(* IEC 61131-3 sources: StandardFunctions/iec61131-st (part 2) *)

(* ---- time_extra_functions.st ---- *)
(********************
*
* Concatenates DATE and TOD to DT
*
*********************)
@EXTERNAL
FUNCTION CONCAT_DATE_TOD : DT
VAR_INPUT
	date_input : DATE;
	tod_input : TOD;
END_VAR
END_FUNCTION

(********************
*
* Concatenates DATE and LTOD to DT
*
*********************)
FUNCTION CONCAT_DATE_LTOD : DT
VAR_INPUT
	date_input : DATE;
	tod_input : LTOD;
END_VAR
	CONCAT_DATE_LTOD := CONCAT_DATE_TOD(date_input, tod_input);
END_FUNCTION

(********************
*
* Concatenates year, month and day of type ANY_INT to DATE
*
*********************)
@EXTERNAL
FUNCTION CONCAT_DATE <T: ANY_INT> : DATE
VAR_INPUT
	year : T;
	month : T;
	day : T;
END_VAR
END_FUNCTION

(********************
*
* Concatenates hour, minute, second, millisecond of type ANY_INT to TOD
*
*********************)
@EXTERNAL
FUNCTION CONCAT_TOD <T: ANY_INT> : TOD
VAR_INPUT
	hour : T;
	minute : T;
	second : T;
	millisecond : T;
END_VAR
END_FUNCTION

(********************
*
* Concatenates hour, minute, second, millisecond of type ANY_INT to LTOD
*
*********************)
FUNCTION CONCAT_LTOD <T: ANY_INT> : LTOD
VAR_INPUT
	hour : T;
	minute : T;
	second : T;
	millisecond : T;
END_VAR
END_FUNCTION

(* Specialized implementation of CONCAT_LTOD for SINT *)
FUNCTION CONCAT_LTOD__SINT : LTOD
VAR_INPUT
	hour : SINT;
	minute : SINT;
	second : SINT;
	millisecond : SINT;
END_VAR
	CONCAT_LTOD__SINT := CONCAT_TOD(hour, minute, second, millisecond);
END_FUNCTION

(* Specialized implementation of CONCAT_LTOD for USINT *)
FUNCTION CONCAT_LTOD__USINT : LTOD
VAR_INPUT
	hour : USINT;
	minute : USINT;
	second : USINT;
	millisecond : USINT;
END_VAR
	CONCAT_LTOD__USINT := CONCAT_TOD(hour, minute, second, millisecond);
END_FUNCTION

(* Specialized implementation of CONCAT_LTOD for INT *)
FUNCTION CONCAT_LTOD__INT : LTOD
VAR_INPUT
	hour : INT;
	minute : INT;
	second : INT;
	millisecond : INT;
END_VAR
	CONCAT_LTOD__INT := CONCAT_TOD(hour, minute, second, millisecond);
END_FUNCTION

(* Specialized implementation of CONCAT_LTOD for UINT *)
FUNCTION CONCAT_LTOD__UINT : LTOD
VAR_INPUT
	hour : UINT;
	minute : UINT;
	second : UINT;
	millisecond : UINT;
END_VAR
	CONCAT_LTOD__UINT := CONCAT_TOD(hour, minute, second, millisecond);
END_FUNCTION

(* Specialized implementation of CONCAT_LTOD for DINT *)
FUNCTION CONCAT_LTOD__DINT : LTOD
VAR_INPUT
	hour : DINT;
	minute : DINT;
	second : DINT;
	millisecond : DINT;
END_VAR
	CONCAT_LTOD__DINT := CONCAT_TOD(hour, minute, second, millisecond);
END_FUNCTION

(* Specialized implementation of CONCAT_LTOD for UDINT *)
FUNCTION CONCAT_LTOD__UDINT : LTOD
VAR_INPUT
	hour : UDINT;
	minute : UDINT;
	second : UDINT;
	millisecond : UDINT;
END_VAR
	CONCAT_LTOD__UDINT := CONCAT_TOD(hour, minute, second, millisecond);
END_FUNCTION

(* Specialized implementation of CONCAT_LTOD for LINT *)
FUNCTION CONCAT_LTOD__LINT : LTOD
VAR_INPUT
	hour : LINT;
	minute : LINT;
	second : LINT;
	millisecond : LINT;
END_VAR
	CONCAT_LTOD__LINT := CONCAT_TOD(hour, minute, second, millisecond);
END_FUNCTION

(* Specialized implementation of CONCAT_LTOD for ULINT *)
FUNCTION CONCAT_LTOD__ULINT : LTOD
VAR_INPUT
	hour : ULINT;
	minute : ULINT;
	second : ULINT;
	millisecond : ULINT;
END_VAR
	CONCAT_LTOD__ULINT := CONCAT_TOD(hour, minute, second, millisecond);
END_FUNCTION

(********************
*
* Concatenates year, month, day, hour, minute, second, millisecond of type ANY_INT to DT
*
*********************)
FUNCTION CONCAT_DT <T: ANY_INT> : DT
VAR_INPUT
	year : T;
	month : T;
	day : T;
	hour : T;
	minute : T;
	second : T;
	millisecond : T;
END_VAR
END_FUNCTION

(* Specialized implementation of CONCAT_DT for INT *)
FUNCTION CONCAT_DT__INT : DT
VAR_INPUT
	year : INT;
	month : INT;
	day : INT;
	hour : INT;
	minute : INT;
	second : INT;
	millisecond : INT;
END_VAR
	CONCAT_DT__INT := CONCAT_DATE_TOD(CONCAT_DATE(year, month, day), CONCAT_TOD(hour, minute, second, millisecond));
END_FUNCTION

(* Specialized implementation of CONCAT_DT for UINT *)
FUNCTION CONCAT_DT__UINT : DT
VAR_INPUT
	year : UINT;
	month : UINT;
	day : UINT;
	hour : UINT;
	minute : UINT;
	second : UINT;
	millisecond : UINT;
END_VAR
	CONCAT_DT__UINT := CONCAT_DATE_TOD(CONCAT_DATE(year, month, day), CONCAT_TOD(hour, minute, second, millisecond));
END_FUNCTION

(* Specialized implementation of CONCAT_DT for DINT *)
FUNCTION CONCAT_DT__DINT : DT
VAR_INPUT
	year : DINT;
	month : DINT;
	day : DINT;
	hour : DINT;
	minute : DINT;
	second : DINT;
	millisecond : DINT;
END_VAR
	CONCAT_DT__DINT := CONCAT_DATE_TOD(CONCAT_DATE(year, month, day), CONCAT_TOD(hour, minute, second, millisecond));
END_FUNCTION

(* Specialized implementation of CONCAT_DT for UDINT *)
FUNCTION CONCAT_DT__UDINT : DT
VAR_INPUT
	year : UDINT;
	month : UDINT;
	day : UDINT;
	hour : UDINT;
	minute : UDINT;
	second : UDINT;
	millisecond : UDINT;
END_VAR
	CONCAT_DT__UDINT := CONCAT_DATE_TOD(CONCAT_DATE(year, month, day), CONCAT_TOD(hour, minute, second, millisecond));
END_FUNCTION

(* Specialized implementation of CONCAT_DT for LINT *)
FUNCTION CONCAT_DT__LINT : DT
VAR_INPUT
	year : LINT;
	month : LINT;
	day : LINT;
	hour : LINT;
	minute : LINT;
	second : LINT;
	millisecond : LINT;
END_VAR
	CONCAT_DT__LINT := CONCAT_DATE_TOD(CONCAT_DATE(year, month, day), CONCAT_TOD(hour, minute, second, millisecond));
END_FUNCTION

(* Specialized implementation of CONCAT_DT for ULINT *)
FUNCTION CONCAT_DT__ULINT : DT
VAR_INPUT
	year : ULINT;
	month : ULINT;
	day : ULINT;
	hour : ULINT;
	minute : ULINT;
	second : ULINT;
	millisecond : ULINT;
END_VAR
	CONCAT_DT__ULINT := CONCAT_DATE_TOD(CONCAT_DATE(year, month, day), CONCAT_TOD(hour, minute, second, millisecond));
END_FUNCTION

(********************
*
* Concatenates year, month, day, hour, minute, second, millisecond of type ANY_INT to LDT
*
*********************)
FUNCTION CONCAT_LDT <T: ANY_INT> : LDT
VAR_INPUT
	year : T;
	month : T;
	day : T;
	hour : T;
	minute : T;
	second : T;
	millisecond : T;
END_VAR
END_FUNCTION

(* Specialized implementation of CONCAT_LDT for INT *)
FUNCTION CONCAT_LDT__INT : LDT
VAR_INPUT
	year : INT;
	month : INT;
	day : INT;
	hour : INT;
	minute : INT;
	second : INT;
	millisecond : INT;
END_VAR
	CONCAT_LDT__INT := CONCAT_DATE_LTOD(CONCAT_DATE(year, month, day), CONCAT_LTOD(hour, minute, second, millisecond));
END_FUNCTION

(* Specialized implementation of CONCAT_LDT for UINT *)
FUNCTION CONCAT_LDT__UINT : LDT
VAR_INPUT
	year : UINT;
	month : UINT;
	day : UINT;
	hour : UINT;
	minute : UINT;
	second : UINT;
	millisecond : UINT;
END_VAR
	CONCAT_LDT__UINT := CONCAT_DATE_LTOD(CONCAT_DATE(year, month, day), CONCAT_LTOD(hour, minute, second, millisecond));
END_FUNCTION

(* Specialized implementation of CONCAT_LDT for DINT *)
FUNCTION CONCAT_LDT__DINT : LDT
VAR_INPUT
	year : DINT;
	month : DINT;
	day : DINT;
	hour : DINT;
	minute : DINT;
	second : DINT;
	millisecond : DINT;
END_VAR
	CONCAT_LDT__DINT := CONCAT_DATE_LTOD(CONCAT_DATE(year, month, day), CONCAT_LTOD(hour, minute, second, millisecond));
END_FUNCTION

(* Specialized implementation of CONCAT_LDT for UDINT *)
FUNCTION CONCAT_LDT__UDINT : LDT
VAR_INPUT
	year : UDINT;
	month : UDINT;
	day : UDINT;
	hour : UDINT;
	minute : UDINT;
	second : UDINT;
	millisecond : UDINT;
END_VAR
	CONCAT_LDT__UDINT := CONCAT_DATE_LTOD(CONCAT_DATE(year, month, day), CONCAT_LTOD(hour, minute, second, millisecond));
END_FUNCTION

(* Specialized implementation of CONCAT_LDT for LINT *)
FUNCTION CONCAT_LDT__LINT : LDT
VAR_INPUT
	year : LINT;
	month : LINT;
	day : LINT;
	hour : LINT;
	minute : LINT;
	second : LINT;
	millisecond : LINT;
END_VAR
	CONCAT_LDT__LINT := CONCAT_DATE_LTOD(CONCAT_DATE(year, month, day), CONCAT_LTOD(hour, minute, second, millisecond));
END_FUNCTION

(* Specialized implementation of CONCAT_LDT for ULINT *)
FUNCTION CONCAT_LDT__ULINT : LDT
VAR_INPUT
	year : ULINT;
	month : ULINT;
	day : ULINT;
	hour : ULINT;
	minute : ULINT;
	second : ULINT;
	millisecond : ULINT;
END_VAR
	CONCAT_LDT__ULINT := CONCAT_DATE_LTOD(CONCAT_DATE(year, month, day), CONCAT_LTOD(hour, minute, second, millisecond));
END_FUNCTION

(********************
*
* Splits DATE into year, month, day of type ANY_INT
*
*********************)
FUNCTION SPLIT_DATE <T: ANY_INT> : INT
VAR_INPUT
	in : DATE;
END_VAR
VAR_OUTPUT
	year : T;
	month : T;
	day : T;
END_VAR
END_FUNCTION

(* Specialized implementation of SPLIT_DATE for INT *)
@EXTERNAL
FUNCTION SPLIT_DATE__INT : INT
VAR_INPUT
	in : DATE;
END_VAR
VAR_OUTPUT
	year : INT;
	month : INT;
	day : INT;
END_VAR
END_FUNCTION

(* Specialized implementation of SPLIT_DATE for UINT *)
@EXTERNAL
FUNCTION SPLIT_DATE__UINT : INT
VAR_INPUT
	in : DATE;
END_VAR
VAR_OUTPUT
	year : UINT;
	month : UINT;
	day : UINT;
END_VAR
END_FUNCTION

(* Specialized implementation of SPLIT_DATE for DINT *)
@EXTERNAL
FUNCTION SPLIT_DATE__DINT : INT
VAR_INPUT
	in : DATE;
END_VAR
VAR_OUTPUT
	year : DINT;
	month : DINT;
	day : DINT;
END_VAR
END_FUNCTION

(* Specialized implementation of SPLIT_DATE for UDINT *)
@EXTERNAL
FUNCTION SPLIT_DATE__UDINT : INT
VAR_INPUT
	in : DATE;
END_VAR
VAR_OUTPUT
	year : UDINT;
	month : UDINT;
	day : UDINT;
END_VAR
END_FUNCTION

(* Specialized implementation of SPLIT_DATE for LINT *)
@EXTERNAL
FUNCTION SPLIT_DATE__LINT : INT
VAR_INPUT
	in : DATE;
END_VAR
VAR_OUTPUT
	year : LINT;
	month : LINT;
	day : LINT;
END_VAR
END_FUNCTION

(* Specialized implementation of SPLIT_DATE for ULINT *)
@EXTERNAL
FUNCTION SPLIT_DATE__ULINT : INT
VAR_INPUT
	in : DATE;
END_VAR
VAR_OUTPUT
	year : ULINT;
	month : ULINT;
	day : ULINT;
END_VAR
END_FUNCTION

(********************
*
* Splits TOD into hour, minute, second, millisecond of type ANY_INT
*
*********************)
FUNCTION SPLIT_TOD <T: ANY_INT> : INT
VAR_INPUT
	in : TOD;
END_VAR
VAR_OUTPUT
	hour : T;
	minute : T;
	second : T;
	millisecond : T;
END_VAR
END_FUNCTION

(* Specialized implementation of SPLIT_TOD for INT *)
@EXTERNAL
FUNCTION SPLIT_TOD__INT : INT
VAR_INPUT
	in : TOD;
END_VAR
VAR_OUTPUT
	hour : INT;
	minute : INT;
	second : INT;
	millisecond : INT;
END_VAR
END_FUNCTION

(* Specialized implementation of SPLIT_TOD for UINT *)
@EXTERNAL
FUNCTION SPLIT_TOD__UINT : INT
VAR_INPUT
	in : TOD;
END_VAR
VAR_OUTPUT
	hour : UINT;
	minute : UINT;
	second : UINT;
	millisecond : UINT;
END_VAR
END_FUNCTION

(* Specialized implementation of SPLIT_TOD for DINT *)
@EXTERNAL
FUNCTION SPLIT_TOD__DINT : INT
VAR_INPUT
	in : TOD;
END_VAR
VAR_OUTPUT
	hour : DINT;
	minute : DINT;
	second : DINT;
	millisecond : DINT;
END_VAR
END_FUNCTION

(* Specialized implementation of SPLIT_TOD for UDINT *)
@EXTERNAL
FUNCTION SPLIT_TOD__UDINT : INT
VAR_INPUT
	in : TOD;
END_VAR
VAR_OUTPUT
	hour : UDINT;
	minute : UDINT;
	second : UDINT;
	millisecond : UDINT;
END_VAR
END_FUNCTION

(* Specialized implementation of SPLIT_TOD for LINT *)
@EXTERNAL
FUNCTION SPLIT_TOD__LINT : INT
VAR_INPUT
	in : TOD;
END_VAR
VAR_OUTPUT
	hour : LINT;
	minute : LINT;
	second : LINT;
	millisecond : LINT;
END_VAR
END_FUNCTION

(* Specialized implementation of SPLIT_TOD for ULINT *)
@EXTERNAL
FUNCTION SPLIT_TOD__ULINT : INT
VAR_INPUT
	in : TOD;
END_VAR
VAR_OUTPUT
	hour : ULINT;
	minute : ULINT;
	second : ULINT;
	millisecond : ULINT;
END_VAR
END_FUNCTION

(********************
*
* Splits LTOD into hour, minute, second, millisecond of type ANY_INT
*
*********************)
FUNCTION SPLIT_LTOD <T: ANY_INT> : INT
VAR_INPUT
	in : LTOD;
END_VAR
VAR_OUTPUT
	hour : T;
	minute : T;
	second : T;
	millisecond : T;
END_VAR
END_FUNCTION

(* Specialized implementation of SPLIT_LTOD for INT *)
FUNCTION SPLIT_LTOD__INT : INT
VAR_INPUT
	in : LTOD;
END_VAR
VAR_OUTPUT
	hour : INT;
	minute : INT;
	second : INT;
	millisecond : INT;
END_VAR
	SPLIT_LTOD__INT := SPLIT_TOD__INT(in, hour, minute, second, millisecond);
END_FUNCTION

(* Specialized implementation of SPLIT_LTOD for UINT *)
FUNCTION SPLIT_LTOD__UINT : INT
VAR_INPUT
	in : LTOD;
END_VAR
VAR_OUTPUT
	hour : UINT;
	minute : UINT;
	second : UINT;
	millisecond : UINT;
END_VAR
	SPLIT_LTOD__UINT := SPLIT_TOD__UINT(in, hour, minute, second, millisecond);
END_FUNCTION

(* Specialized implementation of SPLIT_LTOD for DINT *)
FUNCTION SPLIT_LTOD__DINT : INT
VAR_INPUT
	in : LTOD;
END_VAR
VAR_OUTPUT
	hour : DINT;
	minute : DINT;
	second : DINT;
	millisecond : DINT;
END_VAR
	SPLIT_LTOD__DINT := SPLIT_TOD__DINT(in, hour, minute, second, millisecond);
END_FUNCTION

(* Specialized implementation of SPLIT_LTOD for UDINT *)
FUNCTION SPLIT_LTOD__UDINT : INT
VAR_INPUT
	in : LTOD;
END_VAR
VAR_OUTPUT
	hour : UDINT;
	minute : UDINT;
	second : UDINT;
	millisecond : UDINT;
END_VAR
	SPLIT_LTOD__UDINT := SPLIT_TOD__UDINT(in, hour, minute, second, millisecond);
END_FUNCTION

(* Specialized implementation of SPLIT_LTOD for LINT *)
FUNCTION SPLIT_LTOD__LINT : INT
VAR_INPUT
	in : LTOD;
END_VAR
VAR_OUTPUT
	hour : LINT;
	minute : LINT;
	second : LINT;
	millisecond : LINT;
END_VAR
	SPLIT_LTOD__LINT := SPLIT_TOD__LINT(in, hour, minute, second, millisecond);
END_FUNCTION

(* Specialized implementation of SPLIT_LTOD for ULINT *)
FUNCTION SPLIT_LTOD__ULINT : INT
VAR_INPUT
	in : LTOD;
END_VAR
VAR_OUTPUT
	hour : ULINT;
	minute : ULINT;
	second : ULINT;
	millisecond : ULINT;
END_VAR
	SPLIT_LTOD__ULINT := SPLIT_TOD__ULINT(in, hour, minute, second, millisecond);
END_FUNCTION

(********************
*
* Splits DT into year, month, day, hour, minute, second, millisecond of type ANY_INT
*
*********************)
FUNCTION SPLIT_DT <T: ANY_INT> : INT
VAR_INPUT
	in : DT;
END_VAR
VAR_OUTPUT
	year : T;
	month : T;
	day : T;
	hour : T;
	minute : T;
	second : T;
	millisecond : T;
END_VAR
END_FUNCTION

(* Specialized implementation of SPLIT_DT for INT *)
@EXTERNAL
FUNCTION SPLIT_DT__INT : INT
VAR_INPUT
	in : DT;
END_VAR
VAR_OUTPUT
	year : INT;
	month : INT;
	day : INT;
	hour : INT;
	minute : INT;
	second : INT;
	millisecond : INT;
END_VAR
END_FUNCTION

(* Specialized implementation of SPLIT_DT for UINT *)
@EXTERNAL
FUNCTION SPLIT_DT__UINT : INT
VAR_INPUT
	in : DT;
END_VAR
VAR_OUTPUT
	year : UINT;
	month : UINT;
	day : UINT;
	hour : UINT;
	minute : UINT;
	second : UINT;
	millisecond : UINT;
END_VAR
END_FUNCTION

(* Specialized implementation of SPLIT_DT for DINT *)
@EXTERNAL
FUNCTION SPLIT_DT__DINT : INT
VAR_INPUT
	in : DT;
END_VAR
VAR_OUTPUT
	year : DINT;
	month : DINT;
	day : DINT;
	hour : DINT;
	minute : DINT;
	second : DINT;
	millisecond : DINT;
END_VAR
END_FUNCTION

(* Specialized implementation of SPLIT_DT for UDINT *)
@EXTERNAL
FUNCTION SPLIT_DT__UDINT : INT
VAR_INPUT
	in : DT;
END_VAR
VAR_OUTPUT
	year : UDINT;
	month : UDINT;
	day : UDINT;
	hour : UDINT;
	minute : UDINT;
	second : UDINT;
	millisecond : UDINT;
END_VAR
END_FUNCTION

(* Specialized implementation of SPLIT_DT for LINT *)
@EXTERNAL
FUNCTION SPLIT_DT__LINT : INT
VAR_INPUT
	in : DT;
END_VAR
VAR_OUTPUT
	year : LINT;
	month : LINT;
	day : LINT;
	hour : LINT;
	minute : LINT;
	second : LINT;
	millisecond : LINT;
END_VAR
END_FUNCTION

(* Specialized implementation of SPLIT_DT for ULINT *)
@EXTERNAL
FUNCTION SPLIT_DT__ULINT : INT
VAR_INPUT
	in : DT;
END_VAR
VAR_OUTPUT
	year : ULINT;
	month : ULINT;
	day : ULINT;
	hour : ULINT;
	minute : ULINT;
	second : ULINT;
	millisecond : ULINT;
END_VAR
END_FUNCTION

(********************
*
* Splits LDT into year, month, day, hour, minute, second, millisecond of type ANY_INT
*
*********************)
FUNCTION SPLIT_LDT <T: ANY_INT> : INT
VAR_INPUT
	in : LDT;
END_VAR
VAR_OUTPUT
	year : T;
	month : T;
	day : T;
	hour : T;
	minute : T;
	second : T;
	millisecond : T;
END_VAR
END_FUNCTION

(* Specialized implementation of SPLIT_LDT for INT *)
@EXTERNAL
FUNCTION SPLIT_LDT__INT : INT
VAR_INPUT
	in : LDT;
END_VAR
VAR_OUTPUT
	year : INT;
	month : INT;
	day : INT;
	hour : INT;
	minute : INT;
	second : INT;
	millisecond : INT;
END_VAR
	SPLIT_LDT__INT := SPLIT_DT__INT(in, year, month, day, hour, minute, second, millisecond);
END_FUNCTION

(* Specialized implementation of SPLIT_LDT for UINT *)
@EXTERNAL
FUNCTION SPLIT_LDT__UINT : INT
VAR_INPUT
	in : LDT;
END_VAR
VAR_OUTPUT
	year : UINT;
	month : UINT;
	day : UINT;
	hour : UINT;
	minute : UINT;
	second : UINT;
	millisecond : UINT;
END_VAR
	SPLIT_LDT__UINT := SPLIT_DT__UINT(in, year, month, day, hour, minute, second, millisecond);
END_FUNCTION

(* Specialized implementation of SPLIT_LDT for DINT *)
@EXTERNAL
FUNCTION SPLIT_LDT__DINT : INT
VAR_INPUT
	in : LDT;
END_VAR
VAR_OUTPUT
	year : DINT;
	month : DINT;
	day : DINT;
	hour : DINT;
	minute : DINT;
	second : DINT;
	millisecond : DINT;
END_VAR
	SPLIT_LDT__DINT := SPLIT_DT__DINT(in, year, month, day, hour, minute, second, millisecond);
END_FUNCTION

(* Specialized implementation of SPLIT_LDT for UDINT *)
@EXTERNAL
FUNCTION SPLIT_LDT__UDINT : INT
VAR_INPUT
	in : LDT;
END_VAR
VAR_OUTPUT
	year : UDINT;
	month : UDINT;
	day : UDINT;
	hour : UDINT;
	minute : UDINT;
	second : UDINT;
	millisecond : UDINT;
END_VAR
	SPLIT_LDT__UDINT := SPLIT_DT__UDINT(in, year, month, day, hour, minute, second, millisecond);
END_FUNCTION

(* Specialized implementation of SPLIT_LDT for LINT *)
@EXTERNAL
FUNCTION SPLIT_LDT__LINT : INT
VAR_INPUT
	in : LDT;
END_VAR
VAR_OUTPUT
	year : LINT;
	month : LINT;
	day : LINT;
	hour : LINT;
	minute : LINT;
	second : LINT;
	millisecond : LINT;
END_VAR
	SPLIT_LDT__LINT := SPLIT_DT__LINT(in, year, month, day, hour, minute, second, millisecond);
END_FUNCTION

(* Specialized implementation of SPLIT_LDT for ULINT *)
@EXTERNAL
FUNCTION SPLIT_LDT__ULINT : INT
VAR_INPUT
	in : LDT;
END_VAR
VAR_OUTPUT
	year : ULINT;
	month : ULINT;
	day : ULINT;
	hour : ULINT;
	minute : ULINT;
	second : ULINT;
	millisecond : ULINT;
END_VAR
	SPLIT_LDT__ULINT := SPLIT_DT__ULINT(in, year, month, day, hour, minute, second, millisecond);
END_FUNCTION

(********************
*
* Returns day of week form given DATE in SINT
* 0 -> sunday, 1 -> monday, ..., 6 -> saturday
*
*********************)
@EXTERNAL
FUNCTION DAY_OF_WEEK : SINT
VAR_INPUT
	in : DATE;
END_VAR
END_FUNCTION

(* ---- validation.st ---- *)
(******************************************************************************
Description: Validation function for ANY_REAL
Input:
  - IN: ANY_REAL
Return:
  - FALSE: If input is Not-a-Number(NaN) or infinite(+Inf, -Inf)
  - TRUE: Otherwise
******************************************************************************)
FUNCTION IS_VALID <T: ANY_REAL> : BOOL
VAR_INPUT
	IN : T;
END_VAR
END_FUNCTION

(******************************************************************************
Description: Validation function for ANY_BIT
Validate if the binary representation of the input
would result in a valid BCD representation
Input:
  - IN: ANY_BIT
Return:
  - TRUE: The value of each 4bits representet digit must be between 0-9
  - FALSE: If the value of any 4bits representet digit is higher than 9
******************************************************************************)
FUNCTION IS_VALID_BCD <T: ANY_BIT> : BOOL
VAR_INPUT
	IN : T;
END_VAR
END_FUNCTION

(* ---- bistable_functionblocks.st ---- *)
(******************************************************************************
Description: Bistable function, set dominant
Input:
  - SET1: Dominant input of bistable function.
  - RESET: input of bistable function.
Output:
  - Q1: Result of Bistable function.
Return: Output is used as return
******************************************************************************)
{external}
FUNCTION_BLOCK SR
VAR_INPUT
	SET1: BOOL;
	RESET: BOOL;
END_VAR
VAR_OUTPUT
	Q1: BOOL;
END_VAR
END_FUNCTION_BLOCK

(******************************************************************************
Description: Bistable function, reset dominant.
Input:
  - SET: Bistable input
  - RESET1: Dominmant bistable input.
Output:
  - Q1: Result of bistable function
Return: Output variable used as return value.
******************************************************************************)
{external}
FUNCTION_BLOCK RS
VAR_INPUT
	SET: 	BOOL;
	RESET1: BOOL;
END_VAR
VAR_OUTPUT
	Q1:		BOOL;
END_VAR
END_FUNCTION_BLOCK

(* ---- counters.st ---- *)
(******************************************************************************
Description: Counter up
Input:
  - CU: Count up
  - R: Reset counter to 0
  - PV: Counter limit
Output:
  - Q: Counter reached limit
  - CV: Current counter value
Return: Output is used as return value
******************************************************************************)
{external}
FUNCTION_BLOCK CTU_INT
VAR_INPUT
	CU : BOOL;
	R : BOOL;
	PV : INT;
END_VAR
VAR_OUTPUT
	Q : BOOL;
	CV : INT;
END_VAR
VAR
	M : BOOL;
END_VAR
END_FUNCTION_BLOCK

(******************************************************************************
Description: Counter up
Input:
  - CU: Count up
  - R: Reset counter to 0
  - PV: Counter limit
Output:
  - Q: Counter reached limit
  - CV: Current counter value
Return: Output is used as return value
******************************************************************************)
{external}
FUNCTION_BLOCK CTU_DINT
VAR_INPUT
	CU : BOOL;
	R : BOOL;
	PV : DINT;
END_VAR
VAR_OUTPUT
	Q : BOOL;
	CV : DINT;
END_VAR
VAR
	M : BOOL;
END_VAR
END_FUNCTION_BLOCK

(******************************************************************************
Description: Counter up
Input:
  - CU: Count up
  - R: Reset counter to 0
  - PV: Counter limit
Output:
  - Q: Counter reached limit
  - CV: Current counter value
Return: Output is used as return value
******************************************************************************)
{external}
FUNCTION_BLOCK CTU_UDINT
VAR_INPUT
	CU : BOOL;
	R : BOOL;
	PV : UDINT;
END_VAR
VAR_OUTPUT
	Q : BOOL;
	CV : UDINT;
END_VAR
VAR
	M : BOOL;
END_VAR
END_FUNCTION_BLOCK

(******************************************************************************
Description: Counter up
Input:
  - CU: Count up
  - R: Reset counter to 0
  - PV: Counter limit
Output:
  - Q: Counter reached limit
  - CV: Current counter value
Return: Output is used as return value
******************************************************************************)
{external}
FUNCTION_BLOCK CTU_LINT
VAR_INPUT
	CU : BOOL;
	R : BOOL;
	PV : LINT;
END_VAR
VAR_OUTPUT
	Q : BOOL;
	CV : LINT;
END_VAR
VAR
	M : BOOL;
END_VAR
END_FUNCTION_BLOCK

(******************************************************************************
Description: Counter up
Input:
  - CU: Count up
  - R: Reset counter to 0
  - PV: Counter limit
Output:
  - Q: Counter reached limit
  - CV: Current counter value
Return: Output is used as return value
******************************************************************************)
{external}
FUNCTION_BLOCK CTU_ULINT
VAR_INPUT
	CU : BOOL;
	R : BOOL;
	PV : ULINT;
END_VAR
VAR_OUTPUT
	Q : BOOL;
	CV : ULINT;
END_VAR
VAR
	M : BOOL;
END_VAR
END_FUNCTION_BLOCK

(* ---- timers.st ---- *)
{external}
(******************************************************************************
Description: Timer Pulse
Input:
  - IN: Trigger for Start of the Signal
  - PT: The length of the High-Signal
Output:
  - Q: The pulse
  - ET: The current phase of the High-Signal
Return: Output variables are used for return.
******************************************************************************)
FUNCTION_BLOCK TP
    VAR_INPUT
        IN : BOOL;
        PT : TIME;
    END_VAR
    VAR_OUTPUT
        Q  : BOOL;
        ET : TIME;
    END_VAR
    VAR
        __signal__ : BOOL; (* Value representing the internal signal *)
        __BUFFER__ : ARRAY[1..24] OF BYTE; (* Buffer used for internal implementation *)
    END_VAR
END_FUNCTION_BLOCK

{external}
(******************************************************************************
Description: Timer Pulse
Input:
  - IN: Trigger for Start of the Signal
  - PT: The length of the High-Signal
Output:
  - Q: The pulse
  - ET: The current phase of the High-Signal
Return: Output variables are used for return.
******************************************************************************)
FUNCTION_BLOCK TP_TIME
    VAR_INPUT
        IN : BOOL;
        PT : TIME;
    END_VAR
    VAR_OUTPUT
        Q  : BOOL;
        ET : TIME;
    END_VAR
    VAR
      __signal__ : BOOL; (* Value representing the internal signal *)
      __BUFFER__ : ARRAY[1..24] OF BYTE; (* Buffer used for internal implementation *)
    END_VAR
END_FUNCTION_BLOCK

{external}
(******************************************************************************
Description: Timer Pulse
Input:
  - IN: Trigger for Start of the Signal
  - PT: The length of the High-Signal
Output:
  - Q: The pulse
  - ET: The current phase of the High-Signal
Return: Output variables are used for return.
******************************************************************************)
FUNCTION_BLOCK TP_LTIME
    VAR_INPUT
        IN : BOOL;
        PT : TIME;
    END_VAR
    VAR_OUTPUT
        Q  : BOOL;
        ET : LTIME;
    END_VAR
    VAR
        __signal__ : BOOL; (* Value representing the internal signal *)
        __BUFFER__ : ARRAY[1..24] OF BYTE; (* Buffer used for internal implementation *)
    END_VAR
END_FUNCTION_BLOCK

{external}
(******************************************************************************
Description: Timer on delay.
Input:
  - IN: Starts timer with rising edge, resets timer with falling edge
  - PT: Time to pass, before Q is set
Output:
  - Q: Is TRUE, PT seconds after IN had a rising edge
  - ET: Elapsed time
Return: Output variables are used for return.
******************************************************************************)
FUNCTION_BLOCK TON
VAR_INPUT
	IN: BOOL;
	PT: TIME;
END_VAR
VAR_OUTPUT
	Q: BOOL;
	ET: TIME;
END_VAR
VAR
  __signal__ : BOOL; (* Value representing the internal signal *)
  __BUFFER__ : ARRAY[1..24] OF BYTE; (* Buffer used for internal implementation *)
END_VAR
END_FUNCTION_BLOCK

{external}
(******************************************************************************
Description: Timer on delay.
Input:
  - IN: Starts timer with rising edge, resets timer with falling edge
  - PT: Time to pass, before Q is set
Output:
  - Q: Is TRUE, PT seconds after IN had a rising edge
  - ET: Elapsed time
Return: Output variables are used for return.
******************************************************************************)
FUNCTION_BLOCK TON_TIME
VAR_INPUT
	IN: BOOL;
	PT: TIME;
END_VAR
VAR_OUTPUT
	Q: BOOL;
	ET: TIME;
END_VAR
VAR
  __signal__ : BOOL; (* Value representing the internal signal *)
  __BUFFER__ : ARRAY[1..24] OF BYTE; (* Buffer used for internal implementation *)
END_VAR
END_FUNCTION_BLOCK

{external}
(******************************************************************************
Description: Timer on delay.
Input:
  - IN: Starts timer with rising edge, resets timer with falling edge
  - PT: Time to pass, before Q is set
Output:
  - Q: Is TRUE, PT seconds after IN had a rising edge
  - ET: Elapsed time
Return: Output variables are used for return.
******************************************************************************)
FUNCTION_BLOCK TON_LTIME
VAR_INPUT
	IN: BOOL;
	PT: LTIME;
END_VAR
VAR_OUTPUT
	Q: BOOL;
	ET: TIME;
END_VAR
VAR
  __signal__ : BOOL; (* Value representing the internal signal *)
  __BUFFER__ : ARRAY[1..24] OF BYTE; (* Buffer used for internal implementation *)
END_VAR
END_FUNCTION_BLOCK

(* ---- bit_shift.st ---- *)
(**************************
 *
 * SHL(IN, n)
 *
 * This operator implements a bitwise shift of an operand to the left.
 * IN is shifted by n bit to the left and is filled from the right with zeros.
 *
*************************)
@EXTERNAL FUNCTION SHL<T: ANY_BIT> : T

VAR_INPUT
	IN : T;
	n : DINT;
END_VAR

END_FUNCTION

(**************************
 *
 * SHR(IN, n)
 *
 * This operator implements a bitwise shift of an operand to the right.
 * IN is shifted by n bit to the right.
 * If an unsigned data type is used, filling from the left with zeros ensues.
 * In the case of signed data types, an arithmetic shifting is implemented,
 * i.e. it is filled with the value of the highest bit.
 *
*************************)
@EXTERNAL FUNCTION SHR<T: ANY_BIT> : T

VAR_INPUT
	IN : T;
	n : DINT;
END_VAR

END_FUNCTION

(**************************
 *
 * ROL(IN, n)
 *
 * This operator implements a bitwise rotation of an operand to the left.
 * IN is shifted n-times to the left,
 * whereby the highest bit from the right is again inserted.
 *
*************************)
@EXTERNAL FUNCTION ROL<T : ANY_BIT> : T

VAR_INPUT
	IN : T;
	n : DINT;
END_VAR

END_FUNCTION

(**************************
 *
 * ROR(IN, n)
 *
 * This operator implements a bitwise rotation of an operand to the right.
 * IN is shifted n-times to the right,
 * whereby the lowest bit from the left is again inserted.
 *
*************************)
@EXTERNAL FUNCTION ROR<T: ANY_BIT> : T

VAR_INPUT
	IN : T;
	n : DINT;
END_VAR

END_FUNCTION
